// TIA Portal V20 export
DATA_BLOCK "instFB_AutoCtrl_ABCDE"   // DB4
// stored: InstanceOfName FB_AutoCtrl_ABCDE, InstanceOfType FB
"FB_AutoCtrl_ABCDE"
   // VAR
   //    statExecutePulse : Bool;
   //    statMoveDoneOld : Bool;
   //    statOldStep : Int;
   //    statTargetPos : "UDT_typePoint5";
   //    sRTRIGInitialPath { S7_SetPoint := 'True'} : R_TRIG;
   //    sRTRIGStart { S7_SetPoint := 'True'} : R_TRIG;
   //    sRTRIGStop { S7_SetPoint := 'True'} : R_TRIG;
   //    instMoveLinAbs : MC_MOVELINEARABSOLUTE;
   //    pts { S7_SetPoint := 'True'} : Array[1..5] of "UDT_typePoint5";
   // END_VAR
BEGIN
END_DATA_BLOCK
